// TIA Portal V18 export
FUNCTION "Flowrate adjustment configuration A" : Void   // FC9, LAD
{ S7_Optimized_Access := 'TRUE' }
VERSION : 0.1
// stored: AutoNumber true, IsIECCheckEnabled false, SetENOAutomatically false, UDAEnableTagReadback false
BEGIN

REGION Network 1 (SCL)
   IF "Pump & Flowrate"."Calculated flowrate A without adjustment" <= "Pump & Flowrate".capacity."Pump A" * 0.05 THEN
       "Pump & Flowrate"."fowrate A Adjustment Configuration" := "Flowrate adjustment A".percentage."5%";
   ELSIF "Pump & Flowrate"."Calculated flowrate A without adjustment" <= "Pump & Flowrate".capacity."Pump A" * 0.10 THEN
       "Pump & Flowrate"."fowrate A Adjustment Configuration" := "Flowrate adjustment A".percentage."10%";
   ELSIF "Pump & Flowrate"."Calculated flowrate A without adjustment" <= "Pump & Flowrate".capacity."Pump A" * 0.15 THEN
       "Pump & Flowrate"."fowrate A Adjustment Configuration" := "Flowrate adjustment A".percentage."15%";
   ELSIF "Pump & Flowrate"."Calculated flowrate A without adjustment" <= "Pump & Flowrate".capacity."Pump A" * 0.20 THEN
       "Pump & Flowrate"."fowrate A Adjustment Configuration" := "Flowrate adjustment A".percentage."20%";
   ELSIF "Pump & Flowrate"."Calculated flowrate A without adjustment" <= "Pump & Flowrate".capacity."Pump A" * 0.25 THEN
       "Pump & Flowrate"."fowrate A Adjustment Configuration" := "Flowrate adjustment A".percentage."25%";
   ELSIF "Pump & Flowrate"."Calculated flowrate A without adjustment" <= "Pump & Flowrate".capacity."Pump A" * 0.30 THEN
       "Pump & Flowrate"."fowrate A Adjustment Configuration" := "Flowrate adjustment A".percentage."30%";
   ELSIF "Pump & Flowrate"."Calculated flowrate A without adjustment" <= "Pump & Flowrate".capacity."Pump A" * 0.40 THEN
       "Pump & Flowrate"."fowrate A Adjustment Configuration" := "Flowrate adjustment A".percentage."40%";
   ELSIF "Pump & Flowrate"."Calculated flowrate A without adjustment" <= "Pump & Flowrate".capacity."Pump A" * 0.50 THEN
       "Pump & Flowrate"."fowrate A Adjustment Configuration" := "Flowrate adjustment A".percentage."50%";
   ELSIF "Pump & Flowrate"."Calculated flowrate A without adjustment" <= "Pump & Flowrate".capacity."Pump A" * 0.60 THEN
       "Pump & Flowrate"."fowrate A Adjustment Configuration" := "Flowrate adjustment A".percentage."60%";
   ELSIF "Pump & Flowrate"."Calculated flowrate A without adjustment" <= "Pump & Flowrate".capacity."Pump A" * 0.70 THEN
       "Pump & Flowrate"."fowrate A Adjustment Configuration" := "Flowrate adjustment A".percentage."70%";
   ELSIF "Pump & Flowrate"."Calculated flowrate A without adjustment" <= "Pump & Flowrate".capacity."Pump A" * 0.80 THEN
       "Pump & Flowrate"."fowrate A Adjustment Configuration" := "Flowrate adjustment A".percentage."80%";
   ELSIF "Pump & Flowrate"."Calculated flowrate A without adjustment" <= "Pump & Flowrate".capacity."Pump A" * 0.90 THEN
       "Pump & Flowrate"."fowrate A Adjustment Configuration" := "Flowrate adjustment A".percentage."90%";
   ELSE
       "Pump & Flowrate"."fowrate A Adjustment Configuration" := "Flowrate adjustment A".percentage."100%";
   END_IF;
END_REGION

REGION Network 3: reset alladjustment
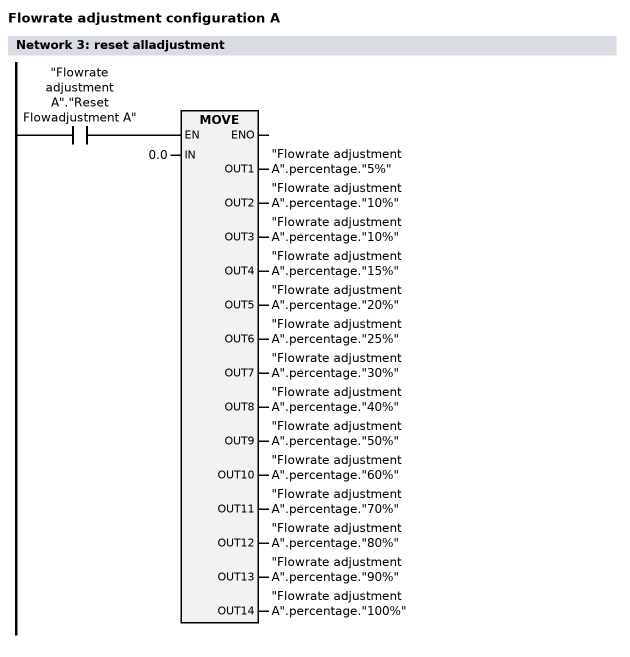
   RUNG wire#powerrail
      Contact( "Flowrate adjustment A"."Reset Flowadjustment A" )
      Move(in := 0.0, out1 => "Flowrate adjustment A".percentage."5%", out2 => "Flowrate adjustment A".percentage."10%", out3 => "Flowrate adjustment A".percentage."10%", out4 => "Flowrate adjustment A".percentage."15%", out5 => "Flowrate adjustment A".percentage."20%", out6 => "Flowrate adjustment A".percentage."25%", out7 => "Flowrate adjustment A".percentage."30%", out8 => "Flowrate adjustment A".percentage."40%", out9 => "Flowrate adjustment A".percentage."50%", out10 => "Flowrate adjustment A".percentage."60%", out11 => "Flowrate adjustment A".percentage."70%", out12 => "Flowrate adjustment A".percentage."80%", out13 => "Flowrate adjustment A".percentage."90%", out14 => "Flowrate adjustment A".percentage."100%")
   END_RUNG
   // the same network as SCL:
   IF "Flowrate adjustment A"."Reset Flowadjustment A" THEN
       "Flowrate adjustment A".percentage."5%" := 0.0;
       "Flowrate adjustment A".percentage."10%" := 0.0;
       "Flowrate adjustment A".percentage."10%" := 0.0;
       "Flowrate adjustment A".percentage."15%" := 0.0;
       "Flowrate adjustment A".percentage."20%" := 0.0;
       "Flowrate adjustment A".percentage."25%" := 0.0;
       "Flowrate adjustment A".percentage."30%" := 0.0;
       "Flowrate adjustment A".percentage."40%" := 0.0;
       "Flowrate adjustment A".percentage."50%" := 0.0;
       "Flowrate adjustment A".percentage."60%" := 0.0;
       "Flowrate adjustment A".percentage."70%" := 0.0;
       "Flowrate adjustment A".percentage."80%" := 0.0;
       "Flowrate adjustment A".percentage."90%" := 0.0;
       "Flowrate adjustment A".percentage."100%" := 0.0;
   END_IF;
END_REGION
END_FUNCTION
